// TwinCAT 3 PLC project DALI_PLC
// ProgramVersion: 3.1.4024.0
// libraries:
//   Tc2_Standard, * (Beckhoff Automation GmbH)
//   Tc2_System, * (Beckhoff Automation GmbH)
//   Tc3_DALI, * (Beckhoff Automation GmbH)
//   Tc3_Module, * (Beckhoff Automation GmbH)
// project tree:
//   / DALI.TcTTO, PlcTask.TcTTO
//   GVLs/ gvlDALI.TcGVL, gvlDALI_State.TcGVL
//   POUs/ MAIN.TcPOU, POU.TcPOU, POU_Comm.TcPOU, WallLight_POU.TcPOU
// real-time tasks:
//   TASK PlcTask: cycle T#10ms, priority 10, ADS port 350
//   TASK DALI: cycle T#2ms, priority 4, ADS port 351
// I/O:
//   DEVICE Device 1 (Beckhoff CCAT)
//   DEVICE Device 2 (CX-BK)
//     Box 1 (CX-BK)
// variable links:
//   DALI_PLC/DALI_PLC Instance <-> Device 2 (CX-BK)/Box 1 (CX-BK)
//     DALI Inputs/gvlDALI.stKL6821InData/aData[{0..3}] <-> Term 8 (KL6821)/Channel 1/Data In {0..3}  (4 links)
//     DALI Inputs/gvlDALI.stKL6821InData/nStatus <-> Term 8 (KL6821)/Channel 1/State
//     DALI Outputs/gvlDALI.stKL6821OutData/aData[{0..3}] <-> Term 8 (KL6821)/Channel 1/Data Out {0..3}  (4 links)
//     DALI Outputs/gvlDALI.stKL6821OutData/nCtrl <-> Term 8 (KL6821)/Channel 1/Ctrl
//     PlcTask Inputs/gvlDALI.bOff <-> Term 3 (KL1809)/Channel 4/Input
//     PlcTask Inputs/gvlDALI.bOff1 <-> Term 5 (KL1408)/Channel 3/Input
//     PlcTask Inputs/gvlDALI.bOff2 <-> Term 4 (KL1809)/Channel 12/Input
//     PlcTask Inputs/gvlDALI.bOff3 <-> Term 4 (KL1809)/Channel 5/Input
//     PlcTask Inputs/gvlDALI.bOff4 <-> Term 4 (KL1809)/Channel 2/Input
//     PlcTask Inputs/gvlDALI.bSwitchOn <-> Term 5 (KL1408)/Channel 6/Input
//     PlcTask Inputs/gvlDALI.bSwitchOn1 <-> Term 3 (KL1809)/Channel 15/Input
//     PlcTask Inputs/gvlDALI.bSwitchOn10 <-> Term 2 (KL1809)/Channel 2/Input
//     PlcTask Inputs/gvlDALI.bSwitchOn11 <-> Term 2 (KL1809)/Channel 3/Input
//     PlcTask Inputs/gvlDALI.bSwitchOn12 <-> Term 2 (KL1809)/Channel 4/Input
//     PlcTask Inputs/gvlDALI.bSwitchOn13 <-> Term 4 (KL1809)/Channel 14/Input
//     PlcTask Inputs/gvlDALI.bSwitchOn14 <-> Term 4 (KL1809)/Channel 13/Input
//     PlcTask Inputs/gvlDALI.bSwitchOn15 <-> Term 2 (KL1809)/Channel 1/Input
//     PlcTask Inputs/gvlDALI.bSwitchOn16 <-> Term 4 (KL1809)/Channel 16/Input
//     PlcTask Inputs/gvlDALI.bSwitchOn17 <-> Term 4 (KL1809)/Channel 15/Input
//     PlcTask Inputs/gvlDALI.bSwitchOn18 <-> Term 5 (KL1408)/Channel 1/Input
//     PlcTask Inputs/gvlDALI.bSwitchOn19 <-> Term 4 (KL1809)/Channel 11/Input
//     PlcTask Inputs/gvlDALI.bSwitchOn2 <-> Term 3 (KL1809)/Channel 12/Input
//     PlcTask Inputs/gvlDALI.bSwitchOn20 <-> Term 4 (KL1809)/Channel 6/Input
//     PlcTask Inputs/gvlDALI.bSwitchOn21 <-> Term 6 (KL1408)/Channel 3/Input
//     PlcTask Inputs/gvlDALI.bSwitchOn22 <-> Term 4 (KL1809)/Channel 8/Input
//     PlcTask Inputs/gvlDALI.bSwitchOn23 <-> Term 4 (KL1809)/Channel 10/Input
//     PlcTask Inputs/gvlDALI.bSwitchOn24 <-> Term 4 (KL1809)/Channel 3/Input
//     PlcTask Inputs/gvlDALI.bSwitchOn25 <-> Term 4 (KL1809)/Channel 1/Input
//     PlcTask Inputs/gvlDALI.bSwitchOn26 <-> Term 2 (KL1809)/Channel 11/Input
//     PlcTask Inputs/gvlDALI.bSwitchOn27 <-> Term 2 (KL1809)/Channel 12/Input
//     PlcTask Inputs/gvlDALI.bSwitchOn28 <-> Term 2 (KL1809)/Channel 10/Input
//     PlcTask Inputs/gvlDALI.bSwitchOn29 <-> Term 2 (KL1809)/Channel 9/Input
//     PlcTask Inputs/gvlDALI.bSwitchOn30 <-> Term 6 (KL1408)/Channel 4/Input
//     PlcTask Inputs/gvlDALI.bSwitchOn4 <-> Term 2 (KL1809)/Channel 14/Input
//     PlcTask Inputs/gvlDALI.bSwitchOn5 <-> Term 3 (KL1809)/Channel 2/Input
//     PlcTask Inputs/gvlDALI.bSwitchOn6 <-> Term 3 (KL1809)/Channel 13/Input
//     PlcTask Inputs/gvlDALI.bSwitchOn7 <-> Term 3 (KL1809)/Channel 14/Input
//     PlcTask Inputs/gvlDALI.bSwitchOn8 <-> Term 3 (KL1809)/Channel 11/Input
//     PlcTask Inputs/gvlDALI.bSwitchOn9 <-> Term 3 (KL1809)/Channel 7/Input
//     PlcTask Outputs/gvlDALI.bRelay0 <-> Term 7 (KL2809)/Channel 3/Output

CONFIGURATION DALI_PLC
    RESOURCE PLC ON TwinCAT3
        TASK DALI(INTERVAL := T#2ms, PRIORITY := 4);
        TASK PlcTask(INTERVAL := T#10ms, PRIORITY := 10);
        PROGRAM POU_Comm WITH DALI : POU_Comm;
        PROGRAM MAIN WITH PlcTask : MAIN;
    END_RESOURCE
END_CONFIGURATION

// ---- GVLs/gvlDALI.TcGVL
{attribute 'qualified_only'}
VAR_GLOBAL
    // ── KL6821 DALI hardware ──────────────────────────────
    stKL6821InData         AT %I* : ST_KL6821InData;
    stKL6821OutData        AT %Q* : ST_KL6821OutData;

    // ── DALI switch inputs (KL1809) ───────────────────────
    bOff                   AT %I* : BOOL;
    bOff1                  AT %I* : BOOL;
    bOff2                  AT %I* : BOOL;
    bOff3                  AT %I* : BOOL;
    bOff4                  AT %I* : BOOL;
    bSwitchOn              AT %I* : BOOL;
    bSwitchOn1             AT %I* : BOOL;
    bSwitchOn2             AT %I* : BOOL;
    bSwitchOn4             AT %I* : BOOL;
    bSwitchOn5             AT %I* : BOOL;
    bSwitchOn6             AT %I* : BOOL;
    bSwitchOn7             AT %I* : BOOL;
    bSwitchOn8             AT %I* : BOOL;
    bSwitchOn9             AT %I* : BOOL;
    bSwitchOn10            AT %I* : BOOL;
    bSwitchOn11            AT %I* : BOOL;
    bSwitchOn12            AT %I* : BOOL;
    bSwitchOn13            AT %I* : BOOL;
    bSwitchOn14            AT %I* : BOOL;
    bSwitchOn15            AT %I* : BOOL;
    bSwitchOn16            AT %I* : BOOL;
    bSwitchOn17            AT %I* : BOOL;
    bSwitchOn18            AT %I* : BOOL;
    bSwitchOn19            AT %I* : BOOL;
    bSwitchOn20            AT %I* : BOOL;
    bSwitchOn21            AT %I* : BOOL;
    bSwitchOn22            AT %I* : BOOL;
    bSwitchOn23            AT %I* : BOOL;
    bSwitchOn24            AT %I* : BOOL;
    bSwitchOn25            AT %I* : BOOL;
    bSwitchOn26            AT %I* : BOOL;
    bSwitchOn27            AT %I* : BOOL;
    bSwitchOn28            AT %I* : BOOL;
    bSwitchOn29            AT %I* : BOOL;
    gButtonLightOn         AT %I* : BOOL;
    gMotionLightOn         AT %I* : BOOL;

    // ── Wall light inputs (KL1819) ────────────────────────
    bSwitchOn30            AT %I* : BOOL;
    bSwitchOn31            AT %I* : BOOL;
    bSwitchOn32            AT %I* : BOOL;
    bSwitchOn33            AT %I* : BOOL;
    bSensor0               AT %I* : BOOL;
    bSensor1               AT %I* : BOOL;
    bSensor2               AT %I* : BOOL;
    bSensor3               AT %I* : BOOL;

    // ── Wall light outputs (KL2809) ───────────────────────
    bRelay0                AT %Q* : BOOL;
    bRelay1                AT %Q* : BOOL;
    bRelay2                AT %Q* : BOOL;
    bRelay3                AT %Q* : BOOL;

    // ── Other non-persistent globals ─────────────────────
    gLightOn               : BOOL;
    bManualMode            : BOOL;

    // ── PyADS bridge: app ↔ PLC control points ────────────
    // Wall relay control (4 physical relays, bRelay0-3) — wired in
    // WallLight_POU below; app writes aPyWallRelay, reads aPyWallRelayState.
    aPyWallRelay           : ARRAY[1..4] OF BOOL;
    aPyWallRelayState      : ARRAY[1..4] OF BOOL;

    // DALI dimmer level control (28 addresses driven by POU.TcPOU) — NOT YET
    // WIRED. POU.TcPOU is a graphical CFC; connect aPySetLevel[N]/aPyLevel[N]
    // to each fbDALI102DimmerNSwitch block's bSetLevel/nLevel input pins, and
    // aPyActualLevel[N] from its nActualLevel output, in the TwinCAT CFC editor.
    aPyLevel               : ARRAY[1..28] OF BYTE;
    aPySetLevel            : ARRAY[1..28] OF BOOL;
    aPyActualLevel         : ARRAY[1..28] OF BYTE;
END_VAR

// ---- GVLs/gvlDALI_State.TcGVL
{attribute 'qualified_only'}
VAR_GLOBAL PERSISTENT
    // ── Wall light states — the ONLY things that need saving ──
    bLightState0           : BOOL;
    bLightState1           : BOOL;
    bLightState2           : BOOL;
    bLightState3           : BOOL;

    bSensorOn0             : BOOL;
    bSensorOn1             : BOOL;
    bSensorOn2             : BOOL;
    bSensorOn3             : BOOL;
END_VAR

// ---- POUs/POU_Comm.TcPOU
PROGRAM POU_Comm
VAR PERSISTENT
	fbKL6821Communication : FB_KL6821Communication; 
	
	bInitialise			  : BOOL;
END_VAR

fbKL6821Communication(
    bInitialise := bInitialise,
    stInData := gvlDALI.stKL6821InData,
    stOutData := gvlDALI.stKL6821OutData); // FB_KL6821Communication

END_PROGRAM

// ---- POUs/MAIN.TcPOU
PROGRAM MAIN
VAR
    bStartupDone   : BOOL := FALSE;   // runs once on boot
    tonStartDelay  : TON;             // small delay to let DALI bus settle first
END_VAR


POU();
WallLight_POU();

END_PROGRAM

// ---- POUs/POU.TcPOU
PROGRAM POU
VAR
    fbDALI102Off             : FB_DALI102Off(POU_Comm.fbKL6821Communication);
    fbDALI102Off1            : FB_DALI102Off(POU_Comm.fbKL6821Communication);
    fbDALI102Off2            : FB_DALI102Off(POU_Comm.fbKL6821Communication);
    fbDALI102Off3            : FB_DALI102Off(POU_Comm.fbKL6821Communication);
    fbDALI102Dimmer1Switch   : FB_DALI102Dimmer1Switch(POU_Comm.fbKL6821Communication);
    fbDALI102Dimmer2Switch   : FB_DALI102Dimmer1Switch(POU_Comm.fbKL6821Communication);
    fbDALI102Dimmer3Switch   : FB_DALI102Dimmer1Switch(POU_Comm.fbKL6821Communication);
    fbDALI102Dimmer4Switch   : FB_DALI102Dimmer1Switch(POU_Comm.fbKL6821Communication);
    fbDALI102Dimmer5Switch   : FB_DALI102Dimmer1Switch(POU_Comm.fbKL6821Communication);
    fbDALI102Dimmer6Switch   : FB_DALI102Dimmer1Switch(POU_Comm.fbKL6821Communication);
    fbDALI102Dimmer7Switch   : FB_DALI102Dimmer1Switch(POU_Comm.fbKL6821Communication);
    fbDALI102Dimmer8Switch   : FB_DALI102Dimmer1Switch(POU_Comm.fbKL6821Communication);
    fbDALI102Dimmer9Switch   : FB_DALI102Dimmer1Switch(POU_Comm.fbKL6821Communication);
    fbDALI102Dimmer10Switch  : FB_DALI102Dimmer1Switch(POU_Comm.fbKL6821Communication);
    fbDALI102Dimmer11Switch  : FB_DALI102Dimmer1Switch(POU_Comm.fbKL6821Communication);
    fbDALI102Dimmer12Switch  : FB_DALI102Dimmer1Switch(POU_Comm.fbKL6821Communication);
    fbDALI102Dimmer13Switch  : FB_DALI102Dimmer1Switch(POU_Comm.fbKL6821Communication);
    fbDALI102Dimmer14Switch  : FB_DALI102Dimmer1Switch(POU_Comm.fbKL6821Communication);
    fbDALI102Dimmer15Switch  : FB_DALI102Dimmer1Switch(POU_Comm.fbKL6821Communication);
    fbDALI102Dimmer16Switch  : FB_DALI102Dimmer1Switch(POU_Comm.fbKL6821Communication);
    fbDALI102Dimmer17Switch  : FB_DALI102Dimmer1Switch(POU_Comm.fbKL6821Communication);
    fbDALI102Dimmer18Switch  : FB_DALI102Dimmer1Switch(POU_Comm.fbKL6821Communication);
    fbDALI102Dimmer19Switch  : FB_DALI102Dimmer1Switch(POU_Comm.fbKL6821Communication);
    fbDALI102Dimmer20Switch  : FB_DALI102Dimmer1Switch(POU_Comm.fbKL6821Communication);
    fbDALI102Dimmer21Switch  : FB_DALI102Dimmer1Switch(POU_Comm.fbKL6821Communication);
    fbDALI102Dimmer22Switch  : FB_DALI102Dimmer1Switch(POU_Comm.fbKL6821Communication);
    fbDALI102Dimmer23Switch  : FB_DALI102Dimmer1Switch(POU_Comm.fbKL6821Communication);
    fbDALI102Dimmer24Switch  : FB_DALI102Dimmer1Switch(POU_Comm.fbKL6821Communication);
    fbDALI102Dimmer25Switch  : FB_DALI102Dimmer1Switch(POU_Comm.fbKL6821Communication);
    fbDALI102Dimmer26Switch  : FB_DALI102Dimmer1Switch(POU_Comm.fbKL6821Communication);
    fbDALI102Dimmer27Switch  : FB_DALI102Dimmer1Switch(POU_Comm.fbKL6821Communication);
    fbDALI102Dimmer28Switch  : FB_DALI102Dimmer1Switch(POU_Comm.fbKL6821Communication);
    bInitialize              : BOOL := FALSE;
    motionSensor             : BOOL;
    bRecallMaxLevel          : BOOL;
    bRecallMinLevel          : BOOL;
    bToggle                  : BOOL;
    bGoToScene               : BOOL;
    nScene                   : BYTE;
    bSetLevel                : BOOL;
    nLevel                   : BYTE := 254;
    nLevelMemoryMode         : BYTE := 254;
    nReferenceDeviceAddress  : BYTE;
    tCycleActualLevel        : TIME := T#5S;
    nOptions                 : DWORD := 0;
    nActualLevel             : BYTE;
END_VAR

fbDALI102Dimmer1Switch(
    bInitialize := bInitialize,
    nAddress := 14,
    eAddressType := E_DALIAddressType.Short,
    bSwitch := gvlDALI.bSwitchOn,
    bRecallMaxLevel := bRecallMaxLevel,
    bRecallMinLevel := bRecallMinLevel,
    bSetLevel := bSetLevel,
    nLevel := nLevel,
    nLevelMemoryMode := nLevelMemoryMode,
    tCycleActualLevel := tCycleActualLevel,
    nOptions := nOptions); // FB_DALI102Dimmer1Switch
nActualLevel := fbDALI102Dimmer18Switch.nActualLevel;
fbDALI102Off(
    bStart := gvlDALI.bOff,
    nAddress := 0,
    eAddressType := E_DALIAddressType.Group,
    eCommandPriority := E_DALICommandPriority.High); // FB_DALI102Off
nActualLevel := fbDALI102Dimmer8Switch.nActualLevel;
nActualLevel := fbDALI102Dimmer25Switch.nActualLevel;
fbDALI102Dimmer6Switch(
    bInitialize := bInitialize,
    nAddress := 3,
    eAddressType := E_DALIAddressType.Short,
    bSwitch := gvlDALI.bSwitchOn6,
    bRecallMaxLevel := bRecallMaxLevel,
    bRecallMinLevel := bRecallMinLevel,
    bSetLevel := bSetLevel,
    nLevel := nLevel,
    nLevelMemoryMode := nLevelMemoryMode,
    tCycleActualLevel := tCycleActualLevel,
    nOptions := nOptions); // FB_DALI102Dimmer1Switch
fbDALI102Dimmer24Switch(
    bInitialize := bInitialize,
    nAddress := 15,
    eAddressType := E_DALIAddressType.Short,
    bSwitch := gvlDALI.bSwitchOn25,
    bRecallMaxLevel := bRecallMaxLevel,
    bRecallMinLevel := bRecallMinLevel,
    bSetLevel := bSetLevel,
    nLevel := nLevel,
    nLevelMemoryMode := nLevelMemoryMode,
    tCycleActualLevel := tCycleActualLevel,
    nOptions := nOptions); // FB_DALI102Dimmer1Switch
fbDALI102Dimmer23Switch(
    bInitialize := bInitialize,
    nAddress := 13,
    eAddressType := E_DALIAddressType.Short,
    bSwitch := gvlDALI.bSwitchOn24,
    bRecallMaxLevel := bRecallMaxLevel,
    bRecallMinLevel := bRecallMinLevel,
    bSetLevel := bSetLevel,
    nLevel := nLevel,
    nLevelMemoryMode := nLevelMemoryMode,
    tCycleActualLevel := tCycleActualLevel,
    nOptions := nOptions); // FB_DALI102Dimmer1Switch
fbDALI102Dimmer21Switch(
    bInitialize := bInitialize,
    nAddress := 15,
    eAddressType := E_DALIAddressType.Short,
    bSwitch := gvlDALI.bSwitchOn22,
    bRecallMaxLevel := bRecallMaxLevel,
    bRecallMinLevel := bRecallMinLevel,
    bSetLevel := bSetLevel,
    nLevel := nLevel,
    nLevelMemoryMode := nLevelMemoryMode,
    tCycleActualLevel := tCycleActualLevel,
    nOptions := nOptions); // FB_DALI102Dimmer1Switch
fbDALI102Dimmer7Switch(
    bInitialize := bInitialize,
    nAddress := 1,
    eAddressType := E_DALIAddressType.Group,
    bSwitch := gvlDALI.bSwitchOn7,
    bRecallMaxLevel := bRecallMaxLevel,
    bRecallMinLevel := bRecallMinLevel,
    bSetLevel := bSetLevel,
    nLevel := nLevel,
    nLevelMemoryMode := nLevelMemoryMode,
    tCycleActualLevel := tCycleActualLevel,
    nOptions := nOptions); // FB_DALI102Dimmer1Switch
fbDALI102Dimmer15Switch(
    bInitialize := bInitialize,
    nAddress := 11,
    eAddressType := E_DALIAddressType.Short,
    bSwitch := gvlDALI.bSwitchOn17,
    bRecallMaxLevel := bRecallMaxLevel,
    bRecallMinLevel := bRecallMinLevel,
    bSetLevel := bSetLevel,
    nLevel := nLevel,
    nLevelMemoryMode := nLevelMemoryMode,
    tCycleActualLevel := tCycleActualLevel,
    nOptions := nOptions); // FB_DALI102Dimmer1Switch
nActualLevel := fbDALI102Dimmer24Switch.nActualLevel;
nActualLevel := fbDALI102Dimmer23Switch.nActualLevel;
fbDALI102Dimmer25Switch(
    bInitialize := bInitialize,
    nAddress := 1,
    eAddressType := E_DALIAddressType.Short,
    bSwitch := gvlDALI.bSwitchOn26,
    bRecallMaxLevel := bRecallMaxLevel,
    bRecallMinLevel := bRecallMinLevel,
    bSetLevel := bSetLevel,
    nLevel := nLevel,
    nLevelMemoryMode := nLevelMemoryMode,
    tCycleActualLevel := tCycleActualLevel,
    nOptions := nOptions); // FB_DALI102Dimmer1Switch
fbDALI102Dimmer26Switch(
    bInitialize := bInitialize,
    nAddress := 10,
    eAddressType := E_DALIAddressType.Short,
    bSwitch := gvlDALI.bSwitchOn27,
    bRecallMaxLevel := bRecallMaxLevel,
    bRecallMinLevel := bRecallMinLevel,
    bSetLevel := bSetLevel,
    nLevel := nLevel,
    nLevelMemoryMode := nLevelMemoryMode,
    tCycleActualLevel := tCycleActualLevel,
    nOptions := nOptions); // FB_DALI102Dimmer1Switch
fbDALI102Dimmer27Switch(
    bInitialize := bInitialize,
    nAddress := 6,
    eAddressType := E_DALIAddressType.Short,
    bSwitch := gvlDALI.bSwitchOn28,
    bRecallMaxLevel := bRecallMaxLevel,
    bRecallMinLevel := bRecallMinLevel,
    bSetLevel := bSetLevel,
    nLevel := nLevel,
    nLevelMemoryMode := nLevelMemoryMode,
    tCycleActualLevel := tCycleActualLevel,
    nOptions := nOptions); // FB_DALI102Dimmer1Switch
fbDALI102Dimmer28Switch(
    bInitialize := bInitialize,
    nAddress := 3,
    eAddressType := E_DALIAddressType.Short,
    bSwitch := gvlDALI.bSwitchOn29,
    bRecallMaxLevel := bRecallMaxLevel,
    bRecallMinLevel := bRecallMinLevel,
    bSetLevel := bSetLevel,
    nLevel := nLevel,
    nLevelMemoryMode := nLevelMemoryMode,
    tCycleActualLevel := tCycleActualLevel,
    nOptions := nOptions); // FB_DALI102Dimmer1Switch
nActualLevel := fbDALI102Dimmer22Switch.nActualLevel;
nActualLevel := fbDALI102Dimmer26Switch.nActualLevel;
nActualLevel := fbDALI102Dimmer27Switch.nActualLevel;
nActualLevel := fbDALI102Dimmer28Switch.nActualLevel;
fbDALI102Dimmer10Switch(
    bInitialize := bInitialize,
    nAddress := 4,
    eAddressType := E_DALIAddressType.Short,
    bSwitch := gvlDALI.bSwitchOn10,
    bRecallMaxLevel := bRecallMaxLevel,
    bRecallMinLevel := bRecallMinLevel,
    bSetLevel := bSetLevel,
    nLevel := nLevel,
    nLevelMemoryMode := nLevelMemoryMode,
    tCycleActualLevel := tCycleActualLevel,
    nOptions := nOptions); // FB_DALI102Dimmer1Switch
fbDALI102Dimmer11Switch(
    bInitialize := bInitialize,
    nAddress := 11,
    eAddressType := E_DALIAddressType.Short,
    bSwitch := gvlDALI.bSwitchOn11,
    bRecallMaxLevel := bRecallMaxLevel,
    bRecallMinLevel := bRecallMinLevel,
    bSetLevel := bSetLevel,
    nLevel := nLevel,
    nLevelMemoryMode := nLevelMemoryMode,
    tCycleActualLevel := tCycleActualLevel,
    nOptions := nOptions); // FB_DALI102Dimmer1Switch
fbDALI102Dimmer16Switch(
    bInitialize := bInitialize,
    nAddress := 5,
    eAddressType := E_DALIAddressType.Short,
    bSwitch := gvlDALI.bSwitchOn18,
    bRecallMaxLevel := bRecallMaxLevel,
    bRecallMinLevel := bRecallMinLevel,
    bSetLevel := bSetLevel,
    nLevel := nLevel,
    nLevelMemoryMode := nLevelMemoryMode,
    tCycleActualLevel := tCycleActualLevel,
    nOptions := nOptions); // FB_DALI102Dimmer1Switch
fbDALI102Dimmer14Switch(
    bInitialize := bInitialize,
    nAddress := 4,
    eAddressType := E_DALIAddressType.Short,
    bSwitch := gvlDALI.bSwitchOn16,
    bRecallMaxLevel := bRecallMaxLevel,
    bRecallMinLevel := bRecallMinLevel,
    bSetLevel := bSetLevel,
    nLevel := nLevel,
    nLevelMemoryMode := nLevelMemoryMode,
    tCycleActualLevel := tCycleActualLevel,
    nOptions := nOptions); // FB_DALI102Dimmer1Switch
nActualLevel := fbDALI102Dimmer16Switch.nActualLevel;
nActualLevel := fbDALI102Dimmer9Switch.nActualLevel;
nActualLevel := fbDALI102Dimmer10Switch.nActualLevel;
nActualLevel := fbDALI102Dimmer11Switch.nActualLevel;
nActualLevel := fbDALI102Dimmer14Switch.nActualLevel;
nActualLevel := fbDALI102Dimmer15Switch.nActualLevel;
fbDALI102Dimmer17Switch(
    bInitialize := bInitialize,
    nAddress := 4,
    eAddressType := E_DALIAddressType.Short,
    bSwitch := gvlDALI.bSwitchOn13,
    bRecallMaxLevel := bRecallMaxLevel,
    bRecallMinLevel := bRecallMinLevel,
    bSetLevel := bSetLevel,
    nLevel := nLevel,
    nLevelMemoryMode := nLevelMemoryMode,
    tCycleActualLevel := tCycleActualLevel,
    nOptions := nOptions); // FB_DALI102Dimmer1Switch
fbDALI102Dimmer22Switch(
    bInitialize := bInitialize,
    nAddress := 15,
    eAddressType := E_DALIAddressType.Short,
    bSwitch := gvlDALI.bSwitchOn23,
    bRecallMaxLevel := bRecallMaxLevel,
    bRecallMinLevel := bRecallMinLevel,
    bSetLevel := bSetLevel,
    nLevel := nLevel,
    nLevelMemoryMode := nLevelMemoryMode,
    tCycleActualLevel := tCycleActualLevel,
    nOptions := nOptions); // FB_DALI102Dimmer1Switch
fbDALI102Dimmer19Switch(
    bInitialize := bInitialize,
    nAddress := 5,
    eAddressType := E_DALIAddressType.Short,
    bSwitch := gvlDALI.bSwitchOn19,
    bRecallMaxLevel := bRecallMaxLevel,
    bRecallMinLevel := bRecallMinLevel,
    bSetLevel := bSetLevel,
    nLevel := nLevel,
    nLevelMemoryMode := nLevelMemoryMode,
    tCycleActualLevel := tCycleActualLevel,
    nOptions := nOptions); // FB_DALI102Dimmer1Switch
nActualLevel := fbDALI102Dimmer21Switch.nActualLevel;
nActualLevel := fbDALI102Dimmer17Switch.nActualLevel;
nActualLevel := fbDALI102Dimmer19Switch.nActualLevel;
fbDALI102Dimmer8Switch(
    bInitialize := bInitialize,
    nAddress := 1,
    eAddressType := E_DALIAddressType.Short,
    bSwitch := gvlDALI.bSwitchOn8,
    bRecallMaxLevel := bRecallMaxLevel,
    bRecallMinLevel := bRecallMinLevel,
    bSetLevel := bSetLevel,
    nLevel := nLevel,
    nLevelMemoryMode := nLevelMemoryMode,
    tCycleActualLevel := tCycleActualLevel,
    nOptions := nOptions); // FB_DALI102Dimmer1Switch
fbDALI102Dimmer3Switch(
    bInitialize := bInitialize,
    nAddress := 0,
    eAddressType := E_DALIAddressType.Short,
    bSwitch := gvlDALI.bSwitchOn2,
    bRecallMaxLevel := bRecallMaxLevel,
    bRecallMinLevel := bRecallMinLevel,
    bSetLevel := bSetLevel,
    nLevel := nLevel,
    nLevelMemoryMode := nLevelMemoryMode,
    tCycleActualLevel := tCycleActualLevel,
    nOptions := nOptions); // FB_DALI102Dimmer1Switch
nActualLevel := fbDALI102Dimmer1Switch.nActualLevel;
nActualLevel := fbDALI102Dimmer6Switch.nActualLevel;
fbDALI102Dimmer20Switch(
    bInitialize := bInitialize,
    nAddress := 13,
    eAddressType := E_DALIAddressType.Short,
    bSwitch := gvlDALI.bSwitchOn20,
    bRecallMaxLevel := bRecallMaxLevel,
    bRecallMinLevel := bRecallMinLevel,
    bSetLevel := bSetLevel,
    nLevel := nLevel,
    nLevelMemoryMode := nLevelMemoryMode,
    tCycleActualLevel := tCycleActualLevel,
    nOptions := nOptions); // FB_DALI102Dimmer1Switch
fbDALI102Dimmer9Switch(
    bInitialize := bInitialize,
    nAddress := 12,
    eAddressType := E_DALIAddressType.Short,
    bSwitch := gvlDALI.bSwitchOn9,
    bRecallMaxLevel := bRecallMaxLevel,
    bRecallMinLevel := bRecallMinLevel,
    bSetLevel := bSetLevel,
    nLevel := nLevel,
    nLevelMemoryMode := nLevelMemoryMode,
    tCycleActualLevel := tCycleActualLevel,
    nOptions := nOptions); // FB_DALI102Dimmer1Switch
fbDALI102Dimmer5Switch(
    bInitialize := bInitialize,
    nAddress := 9,
    eAddressType := E_DALIAddressType.Short,
    bSwitch := gvlDALI.bSwitchOn5,
    bRecallMaxLevel := bRecallMaxLevel,
    bRecallMinLevel := bRecallMinLevel,
    bSetLevel := bSetLevel,
    nLevel := nLevel,
    nLevelMemoryMode := nLevelMemoryMode,
    tCycleActualLevel := tCycleActualLevel,
    nOptions := nOptions); // FB_DALI102Dimmer1Switch
nActualLevel := fbDALI102Dimmer5Switch.nActualLevel;
nActualLevel := fbDALI102Dimmer20Switch.nActualLevel;
fbDALI102Dimmer18Switch(
    bInitialize := bInitialize,
    nAddress := 11,
    eAddressType := E_DALIAddressType.Short,
    bSwitch := gvlDALI.bSwitchOn14,
    bRecallMaxLevel := bRecallMaxLevel,
    bRecallMinLevel := bRecallMinLevel,
    bSetLevel := bSetLevel,
    nLevel := nLevel,
    nLevelMemoryMode := nLevelMemoryMode,
    tCycleActualLevel := tCycleActualLevel,
    nOptions := nOptions); // FB_DALI102Dimmer1Switch
fbDALI102Off3(
    bStart := gvlDALI.bOff4,
    nAddress := 0,
    eAddressType := E_DALIAddressType.Group,
    eCommandPriority := E_DALICommandPriority.High); // FB_DALI102Off
nActualLevel := fbDALI102Dimmer7Switch.nActualLevel;
fbDALI102Dimmer4Switch(
    bInitialize := bInitialize,
    nAddress := 2,
    eAddressType := E_DALIAddressType.Short,
    bSwitch := gvlDALI.bSwitchOn4,
    bRecallMaxLevel := bRecallMaxLevel,
    bRecallMinLevel := bRecallMinLevel,
    bSetLevel := bSetLevel,
    nLevel := nLevel,
    nLevelMemoryMode := nLevelMemoryMode,
    tCycleActualLevel := tCycleActualLevel,
    nOptions := nOptions); // FB_DALI102Dimmer1Switch
nActualLevel := fbDALI102Dimmer3Switch.nActualLevel;
nActualLevel := fbDALI102Dimmer4Switch.nActualLevel;
fbDALI102Dimmer12Switch(
    bInitialize := bInitialize,
    nAddress := 5,
    eAddressType := E_DALIAddressType.Short,
    bSwitch := gvlDALI.bSwitchOn12,
    bRecallMaxLevel := bRecallMaxLevel,
    bRecallMinLevel := bRecallMinLevel,
    bSetLevel := bSetLevel,
    nLevel := nLevel,
    nLevelMemoryMode := nLevelMemoryMode,
    tCycleActualLevel := tCycleActualLevel,
    nOptions := nOptions); // FB_DALI102Dimmer1Switch
nActualLevel := fbDALI102Dimmer12Switch.nActualLevel;
fbDALI102Off2(
    bStart := gvlDALI.bOff2,
    nAddress := 0,
    eAddressType := E_DALIAddressType.Group,
    eCommandPriority := E_DALICommandPriority.High); // FB_DALI102Off
// 3 rd button
fbDALI102Off2(
    bStart := gvlDALI.bOff3,
    nAddress := 0,
    eAddressType := E_DALIAddressType.Group,
    eCommandPriority := E_DALICommandPriority.High); // FB_DALI102Off
fbDALI102Dimmer13Switch(
    bInitialize := bInitialize,
    nAddress := 2,
    eAddressType := E_DALIAddressType.Group,
    bSwitch := gvlDALI.bSwitchOn15,
    bRecallMaxLevel := bRecallMaxLevel,
    bRecallMinLevel := bRecallMinLevel,
    bSetLevel := bSetLevel,
    nLevel := nLevel,
    nLevelMemoryMode := nLevelMemoryMode,
    tCycleActualLevel := tCycleActualLevel,
    nOptions := nOptions); // FB_DALI102Dimmer1Switch
nActualLevel := fbDALI102Dimmer13Switch.nActualLevel;
fbDALI102Off1(
    bStart := gvlDALI.bOff1,
    nAddress := 0,
    eAddressType := E_DALIAddressType.Group,
    eCommandPriority := E_DALICommandPriority.High); // FB_DALI102Off
fbDALI102Dimmer2Switch(
    bInitialize := bInitialize,
    nAddress := 7,
    eAddressType := E_DALIAddressType.Short,
    bSwitch := gvlDALI.bSwitchOn1,
    bRecallMaxLevel := bRecallMaxLevel,
    bRecallMinLevel := bRecallMinLevel,
    bSetLevel := bSetLevel,
    nLevel := nLevel,
    nLevelMemoryMode := nLevelMemoryMode,
    tCycleActualLevel := tCycleActualLevel,
    nOptions := nOptions); // FB_DALI102Dimmer1Switch
nActualLevel := fbDALI102Dimmer2Switch.nActualLevel;

END_PROGRAM

// ---- POUs/WallLight_POU.TcPOU
PROGRAM WallLight_POU
VAR CONSTANT
    // How long a manual OFF (button or app) suppresses the presence sensor
    // from immediately turning the light back on. A deliberate "I'm leaving
    // this off" should stick for a while even if the sensor still sees
    // motion; after this window expires, normal automatic behavior resumes.
    cTempOffSuppress : TIME := T#15M;
END_VAR
VAR
    rTrig_Button0  : R_TRIG;
    rTrig_Button1  : R_TRIG;
    rTrig_Button2  : R_TRIG;
    rTrig_Button3  : R_TRIG;
    tOff0          : TON;
    tOff1          : TON;
    tOff2          : TON;
    tOff3          : TON;

    // TRUE while a manual OFF (button or app) is actively suppressing the
    // presence sensor's auto-on for this light.
    bManualOverride0 : BOOL;
    bManualOverride1 : BOOL;
    bManualOverride2 : BOOL;
    bManualOverride3 : BOOL;
    tManualOverride0 : TON;
    tManualOverride1 : TON;
    tManualOverride2 : TON;
    tManualOverride3 : TON;

    // Last-seen value of each aPyWallRelay[N] — used to detect a fresh
    // app command (edge) without fighting the local button/motion logic.
    aPyWallRelayLast : ARRAY[1..4] OF BOOL;
END_VAR

// ============================================================
// LIGHT 1 — three control sources: physical switch, presence
// sensor (bSensor0), phone app (aPyWallRelay[1]).
// ============================================================
// ── App command (PyADS bridge) ───────────────────────────────────────────
IF gvlDALI.aPyWallRelay[1] <> aPyWallRelayLast[1] THEN
    gvlDALI_State.bLightState0 := gvlDALI.aPyWallRelay[1];
    gvlDALI_State.bSensorOn0   := FALSE;
    // App turned it OFF → temporarily suppress the sensor, like a manual
    // switch-off. App turned it ON → clear any suppression immediately.
    bManualOverride0           := NOT gvlDALI.aPyWallRelay[1];
END_IF

// ── Physical switch ───────────────────────────────────────────────────────
rTrig_Button0(CLK := gvlDALI.bSwitchOn30);
IF rTrig_Button0.Q THEN
    gvlDALI_State.bLightState0 := NOT gvlDALI_State.bLightState0;
    gvlDALI_State.bSensorOn0   := FALSE;
    bManualOverride0           := NOT gvlDALI_State.bLightState0;
END_IF

// ── Presence sensor (suppressed during a manual-override window) ────────
IF gvlDALI.bSensor0 AND NOT gvlDALI_State.bLightState0 AND NOT bManualOverride0 THEN
    gvlDALI_State.bLightState0 := TRUE;
    gvlDALI_State.bSensorOn0   := TRUE;
END_IF

// ── Manual-override expiry ───────────────────────────────────────────────
tManualOverride0(IN := bManualOverride0, PT := cTempOffSuppress);
IF tManualOverride0.Q THEN
    bManualOverride0 := FALSE;
END_IF

// ── Sensor-driven auto-off ────────────────────────────────────────────────
tOff0(IN := gvlDALI_State.bSensorOn0, PT := T#10M);
IF tOff0.Q THEN
    gvlDALI_State.bLightState0 := FALSE;
    gvlDALI_State.bSensorOn0   := FALSE;
END_IF
gvlDALI.bRelay0 := gvlDALI_State.bLightState0;

// resync the app-facing tags so next scan's edge check only fires on a
// genuine new command from the app, not on a local button/motion change.
gvlDALI.aPyWallRelay[1]      := gvlDALI_State.bLightState0;
aPyWallRelayLast[1]          := gvlDALI_State.bLightState0;
gvlDALI.aPyWallRelayState[1] := gvlDALI_State.bLightState0;

// ============================================================
// LIGHT 2
// ============================================================
IF gvlDALI.aPyWallRelay[2] <> aPyWallRelayLast[2] THEN
    gvlDALI_State.bLightState1 := gvlDALI.aPyWallRelay[2];
    gvlDALI_State.bSensorOn1   := FALSE;
    bManualOverride1           := NOT gvlDALI.aPyWallRelay[2];
END_IF

rTrig_Button1(CLK := gvlDALI.bSwitchOn31);
IF rTrig_Button1.Q THEN
    gvlDALI_State.bLightState1 := NOT gvlDALI_State.bLightState1;
    gvlDALI_State.bSensorOn1   := FALSE;
    bManualOverride1           := NOT gvlDALI_State.bLightState1;
END_IF

IF gvlDALI.bSensor1 AND NOT gvlDALI_State.bLightState1 AND NOT bManualOverride1 THEN
    gvlDALI_State.bLightState1 := TRUE;
    gvlDALI_State.bSensorOn1   := TRUE;
END_IF

tManualOverride1(IN := bManualOverride1, PT := cTempOffSuppress);
IF tManualOverride1.Q THEN
    bManualOverride1 := FALSE;
END_IF

tOff1(IN := gvlDALI_State.bSensorOn1, PT := T#10M);
IF tOff1.Q THEN
    gvlDALI_State.bLightState1 := FALSE;
    gvlDALI_State.bSensorOn1   := FALSE;
END_IF
gvlDALI.bRelay1 := gvlDALI_State.bLightState1;

gvlDALI.aPyWallRelay[2]      := gvlDALI_State.bLightState1;
aPyWallRelayLast[2]          := gvlDALI_State.bLightState1;
gvlDALI.aPyWallRelayState[2] := gvlDALI_State.bLightState1;

// ============================================================
// LIGHT 3
// ============================================================
IF gvlDALI.aPyWallRelay[3] <> aPyWallRelayLast[3] THEN
    gvlDALI_State.bLightState2 := gvlDALI.aPyWallRelay[3];
    gvlDALI_State.bSensorOn2   := FALSE;
    bManualOverride2           := NOT gvlDALI.aPyWallRelay[3];
END_IF

rTrig_Button2(CLK := gvlDALI.bSwitchOn32);
IF rTrig_Button2.Q THEN
    gvlDALI_State.bLightState2 := NOT gvlDALI_State.bLightState2;
    gvlDALI_State.bSensorOn2   := FALSE;
    bManualOverride2           := NOT gvlDALI_State.bLightState2;
END_IF

IF gvlDALI.bSensor2 AND NOT gvlDALI_State.bLightState2 AND NOT bManualOverride2 THEN
    gvlDALI_State.bLightState2 := TRUE;
    gvlDALI_State.bSensorOn2   := TRUE;
END_IF

tManualOverride2(IN := bManualOverride2, PT := cTempOffSuppress);
IF tManualOverride2.Q THEN
    bManualOverride2 := FALSE;
END_IF

tOff2(IN := gvlDALI_State.bSensorOn2, PT := T#10M);
IF tOff2.Q THEN
    gvlDALI_State.bLightState2 := FALSE;
    gvlDALI_State.bSensorOn2   := FALSE;
END_IF
gvlDALI.bRelay2 := gvlDALI_State.bLightState2;

gvlDALI.aPyWallRelay[3]      := gvlDALI_State.bLightState2;
aPyWallRelayLast[3]          := gvlDALI_State.bLightState2;
gvlDALI.aPyWallRelayState[3] := gvlDALI_State.bLightState2;

// ============================================================
// LIGHT 4
// ============================================================
IF gvlDALI.aPyWallRelay[4] <> aPyWallRelayLast[4] THEN
    gvlDALI_State.bLightState3 := gvlDALI.aPyWallRelay[4];
    gvlDALI_State.bSensorOn3   := FALSE;
    bManualOverride3           := NOT gvlDALI.aPyWallRelay[4];
END_IF

rTrig_Button3(CLK := gvlDALI.bSwitchOn33);
IF rTrig_Button3.Q THEN
    gvlDALI_State.bLightState3 := NOT gvlDALI_State.bLightState3;
    gvlDALI_State.bSensorOn3   := FALSE;
    bManualOverride3           := NOT gvlDALI_State.bLightState3;
END_IF

IF gvlDALI.bSensor3 AND NOT gvlDALI_State.bLightState3 AND NOT bManualOverride3 THEN
    gvlDALI_State.bLightState3 := TRUE;
    gvlDALI_State.bSensorOn3   := TRUE;
END_IF

tManualOverride3(IN := bManualOverride3, PT := cTempOffSuppress);
IF tManualOverride3.Q THEN
    bManualOverride3 := FALSE;
END_IF

tOff3(IN := gvlDALI_State.bSensorOn3, PT := T#10M);
IF tOff3.Q THEN
    gvlDALI_State.bLightState3 := FALSE;
    gvlDALI_State.bSensorOn3   := FALSE;
END_IF
gvlDALI.bRelay3 := gvlDALI_State.bLightState3;

gvlDALI.aPyWallRelay[4]      := gvlDALI_State.bLightState3;
aPyWallRelayLast[4]          := gvlDALI_State.bLightState3;
gvlDALI.aPyWallRelayState[4] := gvlDALI_State.bLightState3;

END_PROGRAM
